{attribute addProperty BoxType "EK1100-0000-0018"}
{attribute addProperty Id "Beckhoff_EJ4xxxEK1122Beckhoff_EJ4xxxEK1122_15AA3F2B162A_0001_EJ4002_0000_0017EJ4002_19A75BD911314.125A_0002_EJ4002_0000_0018EJ4002_BF483E0111314.125A_0003_EJ4004_0000_0020EJ4004_9786CACB14518.125A_0004_EJ4008_0000_0020EJ4008_D5FA9EBB20926.125A_0005_EJ4018_0000_0016EJ4018_D5FA9EBB20926.125A_0006_EJ4024_0000_0020EJ4024_9786CACB14518.125A_0007_EJ4132_0000_0019EJ4132_19A75BD911314.125A_0008_EJ4134_0000_0019EJ4134_FEE36ED014518.125A_0009_EJ4134_0000_0020EJ4134_FEE36ED014518.125"}
{attribute addProperty CRC "3023301319"}
{attribute addProperty SizeInBites "1353"}
{attribute addProperty SizeInBytes "169.125"}
TYPE Beckhoff_EJ4xxx_B433EAC7 EXTENDS EK1100_179A0949 :
STRUCT
	{attribute addProperty Name "Beckhoff_EJ4xxxEK1122"}
	Beckhoff_EJ4xxxEK1122 : Beckhoff_EJ4xxxEK1122_15AA3F2B;
	{attribute addProperty Name "A_0001_EJ4002_0000_0017"}
	A_0001_EJ4002_0000_0017 : EJ4002_19A75BD9;
	{attribute addProperty Name "A_0002_EJ4002_0000_0018"}
	A_0002_EJ4002_0000_0018 : EJ4002_BF483E01;
	{attribute addProperty Name "A_0003_EJ4004_0000_0020"}
	A_0003_EJ4004_0000_0020 : EJ4004_9786CACB;
	{attribute addProperty Name "A_0004_EJ4008_0000_0020"}
	A_0004_EJ4008_0000_0020 : EJ4008_D5FA9EBB;
	{attribute addProperty Name "A_0005_EJ4018_0000_0016"}
	A_0005_EJ4018_0000_0016 : EJ4018_D5FA9EBB;
	{attribute addProperty Name "A_0006_EJ4024_0000_0020"}
	A_0006_EJ4024_0000_0020 : EJ4024_9786CACB;
	{attribute addProperty Name "A_0007_EJ4132_0000_0019"}
	A_0007_EJ4132_0000_0019 : EJ4132_19A75BD9;
	{attribute addProperty Name "A_0008_EJ4134_0000_0019"}
	A_0008_EJ4134_0000_0019 : EJ4134_FEE36ED0;
	{attribute addProperty Name "A_0009_EJ4134_0000_0020"}
	A_0009_EJ4134_0000_0020 : EJ4134_FEE36ED0;
END_STRUCT
END_TYPE

(* stored: Version 1.2.0.0, ProductVersion 3.1.4024.9
   DUT Beckhoff_EJ4xxx_B433EAC7: Id {efb2f251-ba66-4769-a9aa-b2ab29798f7e} *)
